// Mitsubishi GX Works2 project: EXAM   PLC: Q03UDV

PROGRAM MAIN
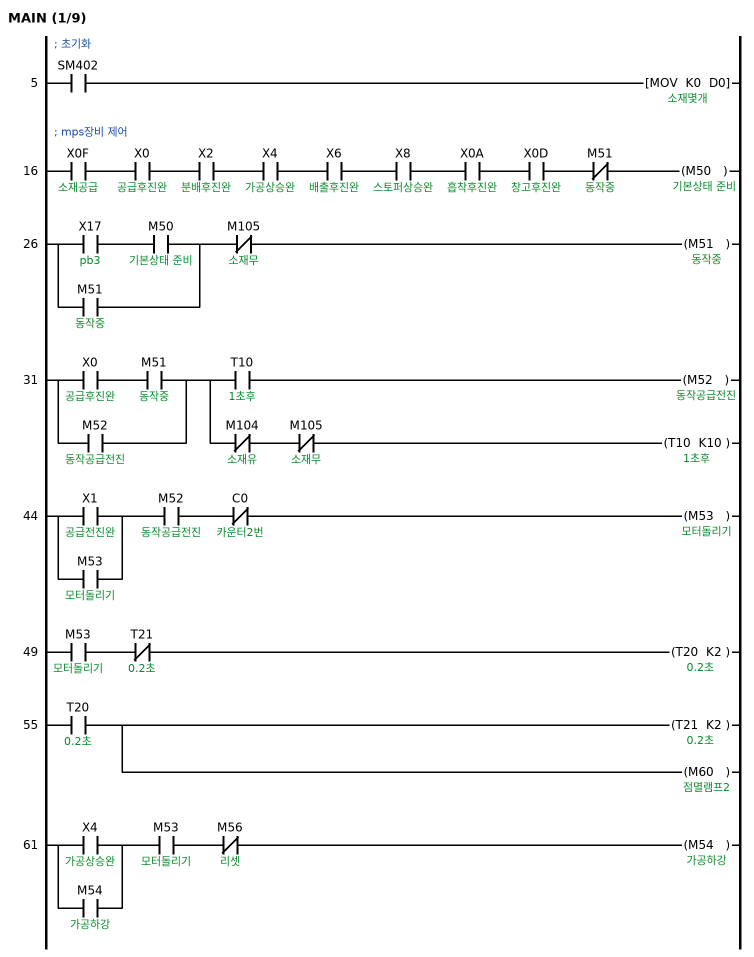
; 초기화
5     LD      SM402
      MOV     K0 D0  ; 소재몇개
; mps장비 제어
16    LD      X0F  ; 소재공급
      AND     X0  ; 공급후진완
      AND     X2  ; 분배후진완
      AND     X4  ; 가공상승완
      AND     X6  ; 배출후진완
      AND     X8  ; 스토퍼상승완
      AND     X0A  ; 흡착후진완
      AND     X0D  ; 창고후진완
      ANI     M51  ; 동작중
      OUT     M50  ; 기본상태 준비
26    LD      X17  ; pb3
      AND     M50  ; 기본상태 준비
      OR      M51  ; 동작중
      ANI     M105  ; 소재무
      OUT     M51  ; 동작중
31    LD      X0  ; 공급후진완
      AND     M51  ; 동작중
      OR      M52  ; 동작공급전진
      MPS
      AND     T10  ; 1초후
      OUT     M52  ; 동작공급전진
      MPP
      ANI     M104  ; 소재유
      ANI     M105  ; 소재무
      OUT     T10 K10  ; 1초후
44    LD      X1  ; 공급전진완
      OR      M53  ; 모터돌리기
      AND     M52  ; 동작공급전진
      ANI     C0  ; 카운터2번
      OUT     M53  ; 모터돌리기
49    LD      M53  ; 모터돌리기
      ANI     T21  ; 0.2초
      OUT     T20 K2  ; 0.2초
55    LD      T20  ; 0.2초
      OUT     T21 K2  ; 0.2초
      OUT     M60  ; 점멸램프2
61    LD      X4  ; 가공상승완
      OR      M54  ; 가공하강
      AND     M53  ; 모터돌리기
      ANI     M56  ; 리셋
      OUT     M54  ; 가공하강
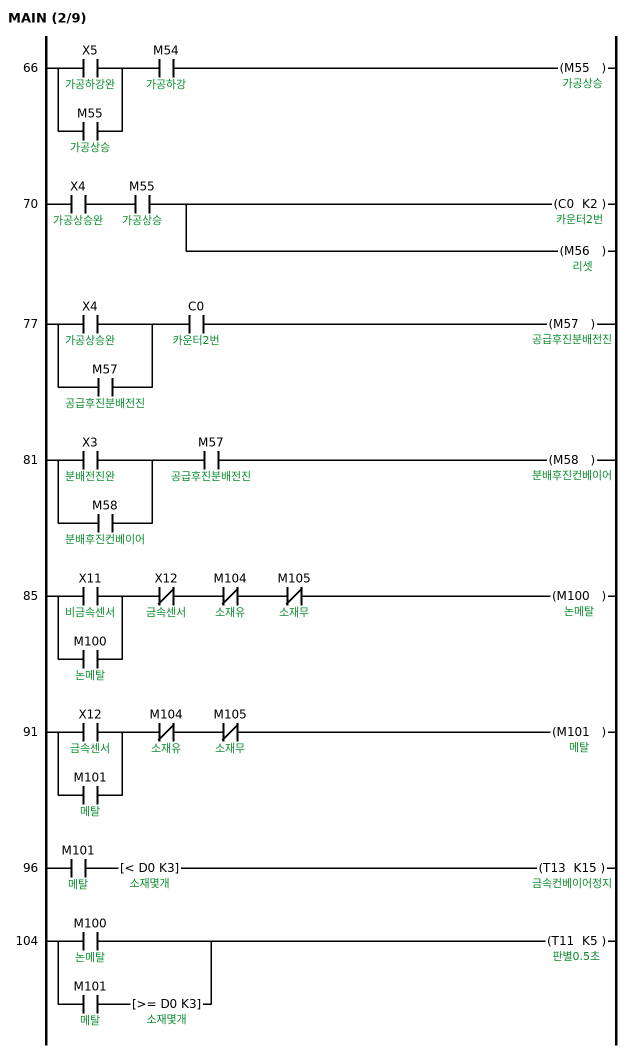
66    LD      X5  ; 가공하강완
      OR      M55  ; 가공상승
      AND     M54  ; 가공하강
      OUT     M55  ; 가공상승
70    LD      X4  ; 가공상승완
      AND     M55  ; 가공상승
      OUT     C0 K2  ; 카운터2번
      OUT     M56  ; 리셋
77    LD      X4  ; 가공상승완
      OR      M57  ; 공급후진분배전진
      AND     C0  ; 카운터2번
      OUT     M57  ; 공급후진분배전진
81    LD      X3  ; 분배전진완
      OR      M58  ; 분배후진컨베이어
      AND     M57  ; 공급후진분배전진
      OUT     M58  ; 분배후진컨베이어
85    LD      X11  ; 비금속센서
      OR      M100  ; 논메탈
      ANI     X12  ; 금속센서
      ANI     M104  ; 소재유
      ANI     M105  ; 소재무
      OUT     M100  ; 논메탈
91    LD      X12  ; 금속센서
      OR      M101  ; 메탈
      ANI     M104  ; 소재유
      ANI     M105  ; 소재무
      OUT     M101  ; 메탈
96    LD      M101  ; 메탈
      AND<    D0 K3  ; 소재몇개
      OUT     T13 K15  ; 금속컨베이어정지
104   LD      M100  ; 논메탈
      LD      M101  ; 메탈
      AND>=   D0 K3  ; 소재몇개
      ORB
      OUT     T11 K5  ; 판별0.5초
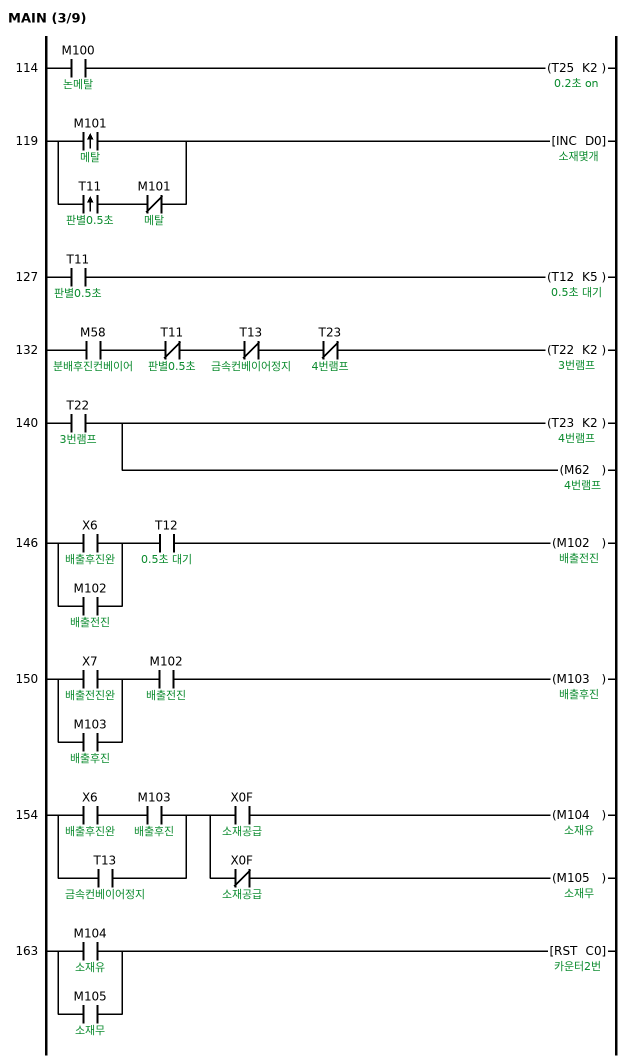
114   LD      M100  ; 논메탈
      OUT     T25 K2  ; 0.2초 on
119   LDP     M101  ; 메탈
      LDP     T11  ; 판별0.5초
      ANI     M101  ; 메탈
      ORB
      INC     D0
127   LD      T11  ; 판별0.5초
      OUT     T12 K5  ; 0.5초 대기
132   LD      M58  ; 분배후진컨베이어
      ANI     T11  ; 판별0.5초
      ANI     T13  ; 금속컨베이어정지
      ANI     T23  ; 4번램프
      OUT     T22 K2  ; 3번램프
140   LD      T22  ; 3번램프
      OUT     T23 K2  ; 4번램프
      OUT     M62  ; 4번램프
146   LD      X6  ; 배출후진완
      OR      M102  ; 배출전진
      AND     T12  ; 0.5초 대기
      OUT     M102  ; 배출전진
150   LD      X7  ; 배출전진완
      OR      M103  ; 배출후진
      AND     M102  ; 배출전진
      OUT     M103  ; 배출후진
154   LD      X6  ; 배출후진완
      AND     M103  ; 배출후진
      OR      T13  ; 금속컨베이어정지
      MPS
      AND     X0F  ; 소재공급
      OUT     M104  ; 소재유
      MPP
      ANI     X0F  ; 소재공급
      OUT     M105  ; 소재무
163   LD      M104  ; 소재유
      OR      M105  ; 소재무
      RST     C0  ; 카운터2번
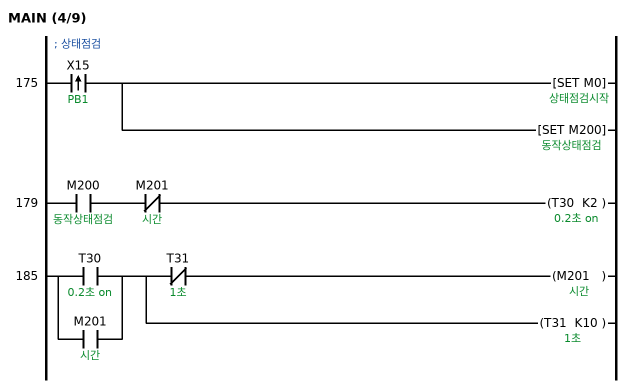
; 상태점검
175   LDP     X15  ; PB1
      SET     M0  ; 상태점검시작
      SET     M200  ; 동작상태점검
179   LD      M200  ; 동작상태점검
      ANI     M201  ; 시간
      OUT     T30 K2  ; 0.2초 on
185   LD      T30  ; 0.2초 on
      OR      M201  ; 시간
      MPS
      ANI     T31  ; 1초
      OUT     M201  ; 시간
      MPP
      OUT     T31 K10  ; 1초
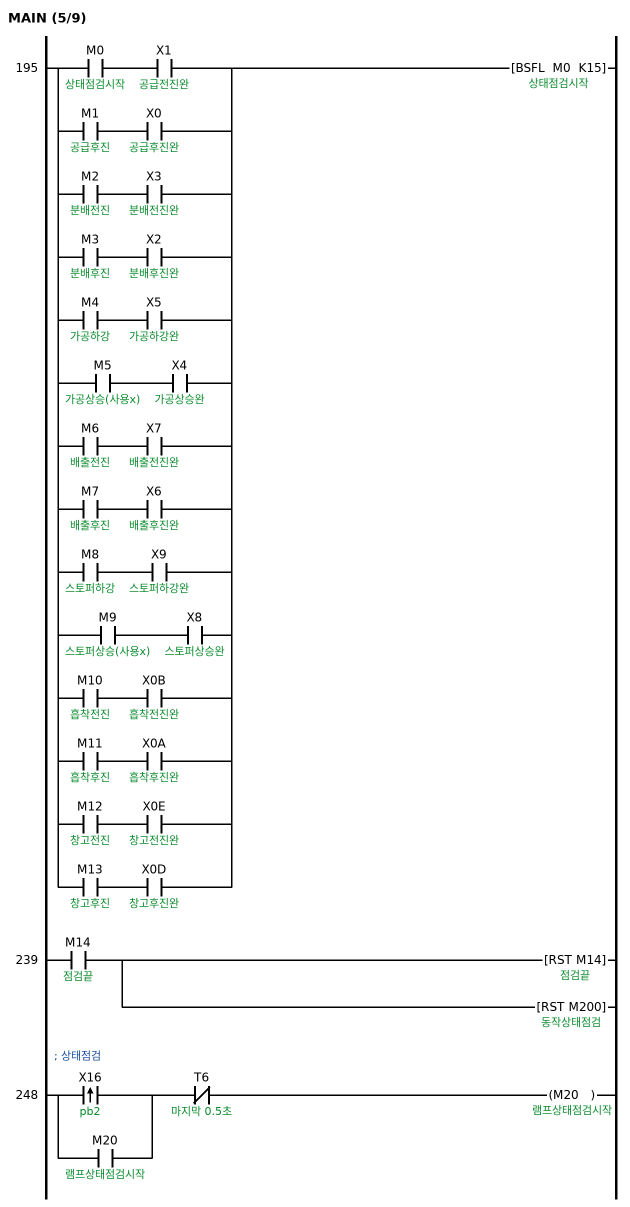
195   LD      M0  ; 상태점검시작
      AND     X1  ; 공급전진완
      LD      M1  ; 공급후진
      AND     X0  ; 공급후진완
      ORB
      LD      M2  ; 분배전진
      AND     X3  ; 분배전진완
      ORB
      LD      M3  ; 분배후진
      AND     X2  ; 분배후진완
      ORB
      LD      M4  ; 가공하강
      AND     X5  ; 가공하강완
      ORB
      LD      M5  ; 가공상승(사용x)
      AND     X4  ; 가공상승완
      ORB
      LD      M6  ; 배출전진
      AND     X7  ; 배출전진완
      ORB
      LD      M7  ; 배출후진
      AND     X6  ; 배출후진완
      ORB
      LD      M8  ; 스토퍼하강
      AND     X9  ; 스토퍼하강완
      ORB
      LD      M9  ; 스토퍼상승(사용x)
      AND     X8  ; 스토퍼상승완
      ORB
      LD      M10  ; 흡착전진
      AND     X0B  ; 흡착전진완
      ORB
      LD      M11  ; 흡착후진
      AND     X0A  ; 흡착후진완
      ORB
      LD      M12  ; 창고전진
      AND     X0E  ; 창고전진완
      ORB
      LD      M13  ; 창고후진
      AND     X0D  ; 창고후진완
      ORB
      BSFL    M0 K15
239   LD      M14  ; 점검끝
      RST     M14  ; 점검끝
      RST     M200  ; 동작상태점검
; 상태점검
248   LDP     X16  ; pb2
      OR      M20  ; 램프상태점검시작
      ANI     T6  ; 마지막 0.5초
      OUT     M20  ; 램프상태점검시작
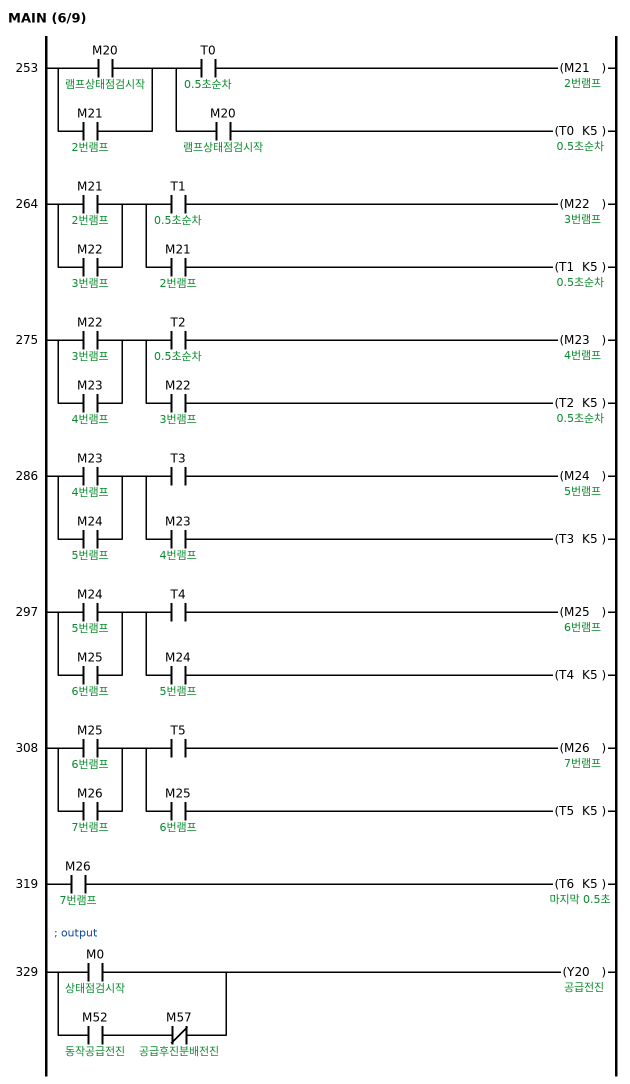
253   LD      M20  ; 램프상태점검시작
      OR      M21  ; 2번램프
      MPS
      AND     T0  ; 0.5초순차
      OUT     M21  ; 2번램프
      MPP
      AND     M20  ; 램프상태점검시작
      OUT     T0 K5  ; 0.5초순차
264   LD      M21  ; 2번램프
      OR      M22  ; 3번램프
      MPS
      AND     T1  ; 0.5초순차
      OUT     M22  ; 3번램프
      MPP
      AND     M21  ; 2번램프
      OUT     T1 K5  ; 0.5초순차
275   LD      M22  ; 3번램프
      OR      M23  ; 4번램프
      MPS
      AND     T2  ; 0.5초순차
      OUT     M23  ; 4번램프
      MPP
      AND     M22  ; 3번램프
      OUT     T2 K5  ; 0.5초순차
286   LD      M23  ; 4번램프
      OR      M24  ; 5번램프
      MPS
      AND     T3
      OUT     M24  ; 5번램프
      MPP
      AND     M23  ; 4번램프
      OUT     T3 K5
297   LD      M24  ; 5번램프
      OR      M25  ; 6번램프
      MPS
      AND     T4
      OUT     M25  ; 6번램프
      MPP
      AND     M24  ; 5번램프
      OUT     T4 K5
308   LD      M25  ; 6번램프
      OR      M26  ; 7번램프
      MPS
      AND     T5
      OUT     M26  ; 7번램프
      MPP
      AND     M25  ; 6번램프
      OUT     T5 K5
319   LD      M26  ; 7번램프
      OUT     T6 K5  ; 마지막 0.5초
; output
329   LD      M0  ; 상태점검시작
      LD      M52  ; 동작공급전진
      ANI     M57  ; 공급후진분배전진
      ORB
      OUT     Y20  ; 공급전진
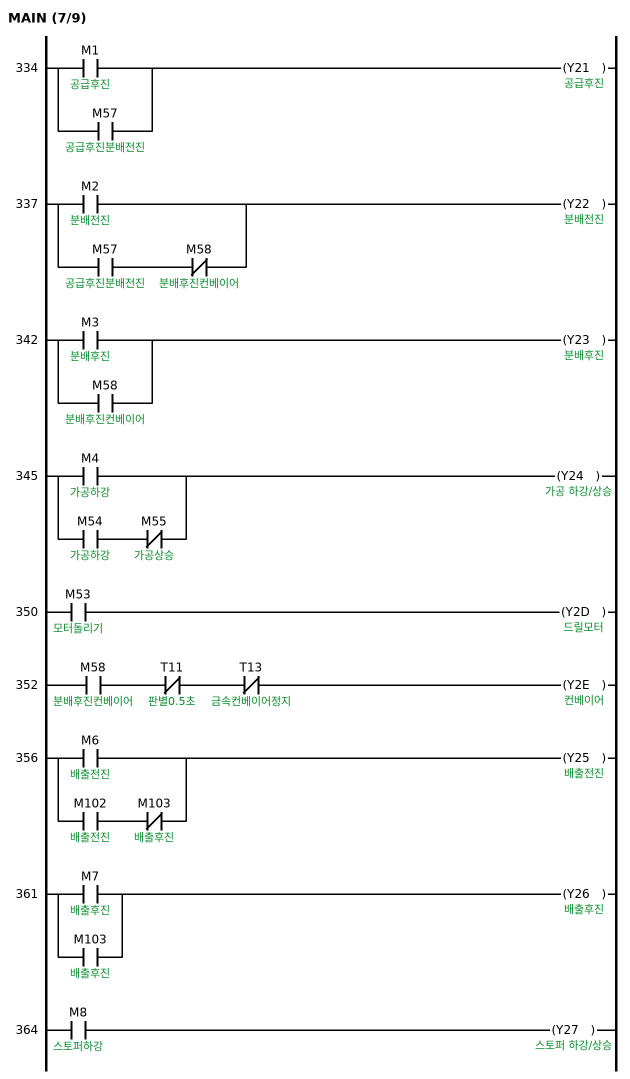
334   LD      M1  ; 공급후진
      OR      M57  ; 공급후진분배전진
      OUT     Y21  ; 공급후진
337   LD      M2  ; 분배전진
      LD      M57  ; 공급후진분배전진
      ANI     M58  ; 분배후진컨베이어
      ORB
      OUT     Y22  ; 분배전진
342   LD      M3  ; 분배후진
      OR      M58  ; 분배후진컨베이어
      OUT     Y23  ; 분배후진
345   LD      M4  ; 가공하강
      LD      M54  ; 가공하강
      ANI     M55  ; 가공상승
      ORB
      OUT     Y24  ; 가공 하강/상승
350   LD      M53  ; 모터돌리기
      OUT     Y2D  ; 드릴모터
352   LD      M58  ; 분배후진컨베이어
      ANI     T11  ; 판별0.5초
      ANI     T13  ; 금속컨베이어정지
      OUT     Y2E  ; 컨베이어
356   LD      M6  ; 배출전진
      LD      M102  ; 배출전진
      ANI     M103  ; 배출후진
      ORB
      OUT     Y25  ; 배출전진
361   LD      M7  ; 배출후진
      OR      M103  ; 배출후진
      OUT     Y26  ; 배출후진
364   LD      M8  ; 스토퍼하강
      OUT     Y27  ; 스토퍼 하강/상승
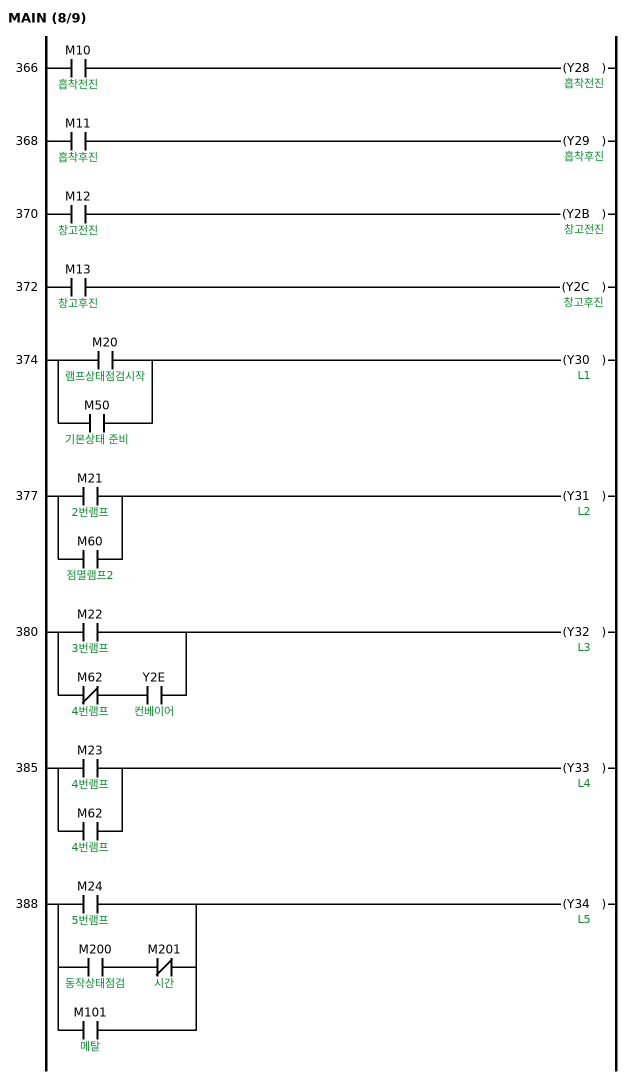
366   LD      M10  ; 흡착전진
      OUT     Y28  ; 흡착전진
368   LD      M11  ; 흡착후진
      OUT     Y29  ; 흡착후진
370   LD      M12  ; 창고전진
      OUT     Y2B  ; 창고전진
372   LD      M13  ; 창고후진
      OUT     Y2C  ; 창고후진
374   LD      M20  ; 램프상태점검시작
      OR      M50  ; 기본상태 준비
      OUT     Y30  ; L1
377   LD      M21  ; 2번램프
      OR      M60  ; 점멸램프2
      OUT     Y31  ; L2
380   LD      M22  ; 3번램프
      LDI     M62  ; 4번램프
      AND     Y2E  ; 컨베이어
      ORB
      OUT     Y32  ; L3
385   LD      M23  ; 4번램프
      OR      M62  ; 4번램프
      OUT     Y33  ; L4
388   LD      M24  ; 5번램프
      LD      M200  ; 동작상태점검
      ANI     M201  ; 시간
      ORB
      OR      M101  ; 메탈
      OUT     Y34  ; L5
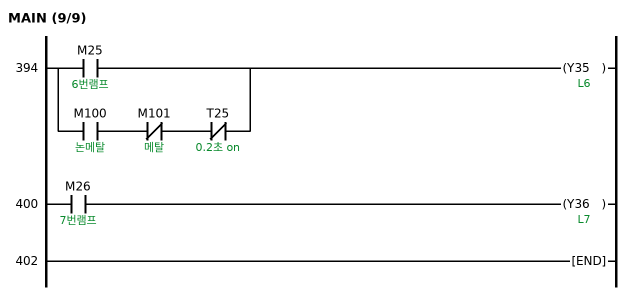
394   LD      M25  ; 6번램프
      LD      M100  ; 논메탈
      ANI     M101  ; 메탈
      ANI     T25  ; 0.2초 on
      ORB
      OUT     Y35  ; L6
400   LD      M26  ; 7번램프
      OUT     Y36  ; L7
402   END
END_PROGRAM

// device comments not shown above
M61  ; 3번램프
C1  ; 확인용
